Staubli VAL3: retain.dtx


